PROGRAM p20_timer
VAR
END_VAR

END_PROGRAM

(* stored: Version 1.1.0.1, ProductVersion 3.1.4024.13
   POU p20_timer: Id {5e4b95fb-c4c9-4cab-ab38-cbb69043119d}, SpecialFunc None *)
